// TwinCAT 3 PLC project PLC
// ProgramVersion: 3.1.4023.0
// libraries:
//   Tc2_Standard, * (Beckhoff Automation GmbH)
//   Tc2_System, * (Beckhoff Automation GmbH)
//   Tc2_Utilities, * (Beckhoff Automation GmbH)
//   Tc3_Module, * (Beckhoff Automation GmbH)
// project tree:
//   Encryption/Blowfish/ FB_Blowfish.TcPOU, P_Blowfish.TcPOU
//   / PlcTask.TcTTO
//   POUs/ MAIN.TcPOU
// real-time tasks:
//   TASK PlcTask: cycle T#10ms, priority 20, ADS port 350

CONFIGURATION PLC
    RESOURCE PLC ON TwinCAT3
        TASK PlcTask(INTERVAL := T#10ms, PRIORITY := 20);
        PROGRAM MAIN WITH PlcTask : MAIN;
    END_RESOURCE
END_CONFIGURATION

// ---- POUs/MAIN.TcPOU
PROGRAM MAIN

// Blowfish test
P_Blowfish();

END_PROGRAM

// ---- Encryption/Blowfish/P_Blowfish.TcPOU
(* 
	Encrypting data with the Blowfish algorithm
	More info: https://www.schneier.com/academic/blowfish/

	original code 
	C by Bruce Schneier	https://www.schneier.com/wp-content/uploads/2015/12/bfsh-sch.zip

	TwinCAT code released under MIT license (https://opensource.org/licenses/MIT)
	Kim Robbens (2022) 	
	
	USAGE:
		* The subkeyfile BLOWFISH.DAT should be placed in the TwinCAT default boot folder. 
		  In most cases this is C:\TwinCAT\3.1\Boot.
		* define instance of FB_BlowFish
		* define a secret key, can be any data type, the max length is 56 bytes / 448 bits
		  as defined in the Blowfish specification
		* initialize the FB_Blowfish instance with the necessary parameters  
			- secret key
			- length of the secret key
			- endianness of the system, TRUE: Eg: Intel, FALSE: Eg: Motorola 
*)
PROGRAM P_Blowfish
VAR
	// Blowfish algorithm
	fbBlowFish			: FB_BlowFish;
	
	// Test secret key
	key 				: T_MAXSTRING := 'TESTKEY';
	
	
	
	(********************  UNIT TESTS  ***********************)
	// Test string to encrypt, its length should be a multiple of 4 bytes
	// real size of a string is [15] + NULL character == 16 !!
	sString				: STRING[15] := 'ABCDEFGHIJKLMNO';	
	nStringLengthOK		: DINT;
	// If the length is nok, an error will be returned with the # of exceeding bytes 
	sStringNOK			: STRING[17] := 'ABCD_EFGH_IJKL_MN';
	nStringLengthNOK	: DINT;

	// Test array to encrypt
	byBytes				: ARRAY[0..7] OF BYTE := [16#11,16#12,16#13,16#14,16#15,16#16,16#0,16#0];
	nArrayLengthOK		: DINT;
	
	// Test lreal
	lr					: LREAL := 123.2231; // be aware of binary notation rounding!
	nlr					: DINT;

	// test lint
	li					: LINT := -12123123412345;
	nli					: DINT;	
	(********************  UNIT TESTS  ***********************)
END_VAR

// Make sure the subkey file blowfish.dat is located in the TwinCAT 3 root boot folder
// eg. C:\TwinCAT\3.1\Boot

// Blowfish implementation test
IF fbBlowFish.bInitialized		THEN
	(********************  UNIT TESTS  ***********************)
	// Any datatype can be used to encrypt, 
	// as long as it real length MOD 8 == 0
	// examples below 
	nStringLengthOK 	:= fbBlowFish.encrypt(sString);		// string length is ok
	nStringLengthOK 	:= fbBlowFish.decrypt(sString);
	nStringLengthNOK 	:= fbBlowFish.encrypt(sStringNOK);	// returns the # of extra characters
	nStringLengthNOK 	:= fbBlowFish.decrypt(sStringNOK);
	nArrayLengthOK 		:= fbBlowFish.encrypt(byBytes);		// test bytes array
	nArrayLengthOK 		:= fbBlowFish.decrypt(byBytes);
	nlr 				:= fbBlowFish.encrypt(lr);			// test lreal
	nlr 				:= fbBlowFish.decrypt(lr);
	nli 				:= fbBlowFish.encrypt(li);			// test lint
	nli 				:= fbBlowFish.decrypt(li);	
	(********************  UNIT TESTS  ***********************)
ELSE	// Initializing
	fbBlowFish(SecretKey:=ADR(key), SecretKeyBytes:=len(key), bLittleEndian:=TRUE);	
END_IF

END_PROGRAM

// ---- Encryption/Blowfish/FB_Blowfish.TcPOU
(* 
	Encrypting data with the Blowfish algorithm, more info below

	original code 
	C by Bruce Schneier	https://www.schneier.com/wp-content/uploads/2015/12/bfsh-sch.zip

	TwinCAT code released under MIT license (https://opensource.org/licenses/MIT)
	Kim Robbens (2022) 
	
	<!HARD LIMITATION
	Due to the limitations of codesys memory allocations,
	it is only possible to encrypt datablocks that have a byte length MOD 8 == 0	
	eg STRING[8] is 9 bytes!!
	See example implementation
	HARD LIMITATION!>
*)
{attribute 'hide_all_locals'}
FUNCTION_BLOCK FB_Blowfish
VAR_INPUT
	SecretKey				: POINTER TO BYTE;	// Make sure that the object is a multiple of 4 bytes!
	SecretKeyBytes			: INT;
	bLittleEndian			: BOOL:=TRUE;	(* TRUE: Eg: Intel, FALSE: Eg: Motorola *)
END_VAR
VAR_OUTPUT
	bBusy                   : BOOL; 	(* TRUE => execution in progress, FALSE => execution idle *)
 	bError                  : BOOL; 	(* TRUE => Error, FALSE => No error *)
	bInitialized			: BOOL;		(* TRUE => initialization of the cipher OK *)
 	nErrorId                : UDINT;	(* Error code *)
END_VAR
VAR
	// Internal selftest results
	bSelfTestEncryptionOK	: BOOL;		(* TRUE => internal encryption selftest OK *)
	bSelfTestDecryptionOK	: BOOL;		(* TRUE => internal decryption selftest OK *)	

	// Local Blowfish state enum
	eBF_State				: (	E_BF_Idle, 
								E_BF_FileOpen, E_BF_FileOpening, E_BF_FileIsOpened, 
								E_BF_P_Array_Read, E_BF_P_Array_IsRead, 
								E_BF_S_Boxes_Read, E_BF_S_Boxes_IsRead, 
								E_BF_FileClose, E_BF_FileClosing, E_BF_FileIsClosed,
								E_BF_SelfTest_Encryption, E_BF_SelfTest_Decryption,
								E_BF_Ready, E_BF_Error);		
	// Local error identification
	eErrorID				: ( E_ERR_NoError,
								E_ERR_SelfTest_Encryption,
								E_ERR_DataLength_NOK);
	// File handling
	hSubKeyFile				: UINT := 0;(* File handle of the subkey file *)
	fbFileOpen              : FB_FileOpen;
	fbFileClose             : FB_FileClose;
	fbFileRead              : FB_FileRead;
	// P-Array and S-Boxes
	_P						: ARRAY[0..N+1] OF UDINT; 		// unsigned long P[N + 2];
	_S						: ARRAY[0..3,0..255] OF UDINT; 	// unsigned long S[4][256];
END_VAR
VAR CONSTANT
	MAXKEYBYTES 			: BYTE := 56;          // 448 bits 
	N               		: BYTE := 16;
	subKeyFilename   		: T_MAXSTRING := 'Blowfish.dat';	
END_VAR
(* 
	Encrypting data with the Blowfish algorithm, info below

	Blowfish is unpatented and license-free, and is available free for all uses.

	Source: https://www.embedded.com/encrypting-data-with-the-blowfish-algorithm/

	Generally speaking, encryption algorithms come in two flavors, symmetric and public key. 
	Symmetric algorithms, such as Blowfish, use the same key for encryption and decryption. 
	Like a password, you have to keep the key secret from everyone except the sender and receiver 
	of the message. 

	Blowfish is a symmetric encryption algorithm, meaning that it uses the same secret key 
	to both encrypt and decrypt messages. 
	Blowfish is also a block cipher, meaning that it divides a message up into fixed length blocks 
	during encryption and decryption. The block length for Blowfish is 64 bits; 
	messages that aren't a multiple of eight bytes in size must be padded.

	Blowfish is public domain, and was designed by Bruce Schneier expressly for use in 
	performance-constrained environments such as embedded systems. 
	It has been extensively analyzed and deemed "reasonably secure" by the cryptographic community. 
	Implementation examples are available from several sources, including the one by Bruce Schneier 
	and the one from Paul Kocher that have been used for creating the TwinCAT compatible version. 
	The original code is available for download at https://www.schneier.com/academic/blowfish/download/

	More info: https://www.schneier.com/academic/blowfish/
	
	port of original code 
	C by Bruce Schneier	https://www.schneier.com/wp-content/uploads/2015/12/bfsh-sch.zip
*)

IF NOT bInitialized		THEN
	initialize(SecretKey, SecretKeyBytes, TRUE);
END_IF

METHOD private _busy
bInitialized	:= FALSE;
bError			:= FALSE;
nErrorID		:= TO_UDINT(E_ERR_NoError);
bBusy 			:= TRUE;
END_METHOD

METHOD PRIVATE _done
bError			:= FALSE;
bBusy 			:= FALSE;
nErrorID		:= TO_UDINT(E_ERR_NoError);
bInitialized	:= TRUE;
END_METHOD

METHOD PRIVATE _error
VAR_INPUT
END_VAR
bBusy 			:= FALSE;
bError			:= TRUE;
END_METHOD

METHOD PRIVATE decipher
VAR_INPUT
	xL					: REFERENCE TO UDINT;
	xR					: REFERENCE TO UDINT;
END_VAR
VAR
	temp				: UDINT;
	i					: INT;
END_VAR
FOR i := N+1 TO 2 BY -1 DO		// for (i = N + 1; i > 1; --i)
	xL		:= xL XOR _P[i];
	xR 	:= F(xL) XOR xR;
	// Exchange xL and xR 
	temp 	:= xL;
	xL 	:= xR;
	xR 	:= temp;
END_FOR

// Exchange xL and xR
temp 		:= xL;
xL 		:= xR;
xR 		:= temp;

xR 		:= xR XOR _P[1];
xL 		:= xL XOR _P[0];
END_METHOD

METHOD PUBLIC decrypt 		: DINT
VAR_INPUT
	data					: ANY;	// !!! Only 8 byte multiple sized BYTE arrays !!!
END_VAR
VAR
	dataL					: UDINT;
	dataR					: UDINT;	
	i						: DINT;	
	nMultiples				: DINT;		// Number of blocks of 4 byte
	bEvenMultiples			: BOOL;		// Number of blocks of 4 byte is even
END_VAR
IF bInitialized 			THEN		// Cipher was initialized
	// Blowfish is a 4/8 byte block cipher
	// so first check the length of the data
	// if the data is no multiple of 4, exit with error
	decrypt					:= data.diSize MOD 4;
	IF decrypt = 0 	AND_THEN data.diSize > 0	THEN
		nMultiples			:= data.diSize / 4;				// Number of blocks
		bEvenMultiples		:= nMultiples MOD 2 = 0;		// Even number of blocks
		FOR i := 0 TO nMultiples-1 BY 2 DO
			dataL				:=
			dataR				:= 16#0;
			memcpy(ADR(dataL), ADR(data.pValue[i*4]), 4);
			IF 	i <	nMultiples-1 OR_ELSE bEvenMultiples THEN
				memcpy(ADR(dataR), ADR(data.pValue[(i+1)*4]), 4);
				decipher(dataL, dataR);
				memcpy(ADR(data.pValue[i*4]), ADR(dataL), 4);				
				memcpy(ADR(data.pValue[(i+1)*4]), ADR(dataR), 4);
			ELSE
				decipher(dataL, dataR);
				memcpy(ADR(data.pValue[i*4]), ADR(dataL), 4);				
			END_IF	
		END_FOR
	ELSE
		nErrorId			:= TO_UDINT(E_ERR_DataLength_NOK);
		_error();		
	END_IF  
ELSE
	initialize(SecretKey, SecretKeyBytes, bLittleEndian);
END_IF
END_METHOD

METHOD PRIVATE encipher
VAR_INPUT
	xL					: REFERENCE TO UDINT;
	xR					: REFERENCE TO UDINT;
END_VAR
VAR
	i					: INT;
	temp				: UDINT;
END_VAR
FOR i := 0 TO N-1 DO				// for (i = 0; i < N; ++i)
	xL		:= xL XOR _P[i];
	xR 		:= F(xL) XOR xR;
	// Exchange xL and xR
	temp 	:= xL;
	xL 		:= xR;
	xR 		:= temp;
END_FOR

// Exchange xL and xR 
temp 		:= xL;
xL 			:= xR;
xR 			:= temp;

xR 			:= xR XOR _P[N];		// Xr = Xr ^ _P[N];
xL 			:= xL XOR _P[N + 1];	// Xl = Xl ^ _P[N + 1];
END_METHOD

METHOD PUBLIC encrypt 		: DINT
VAR_INPUT
	data					: ANY;	// !!! Only 8 byte multiple sized BYTE data !!!
END_VAR
VAR
	dataL					: UDINT;
	dataR					: UDINT;	
	i						: DINT;	
	nMultiples				: DINT;		// Number of blocks of 4 byte
	bEvenMultiples			: BOOL;		// Number of blocks of 4 byte is even
END_VAR
IF bInitialized 			THEN		// Cipher was initialized
	// Blowfish is a 4/8 byte block cipher
	// so first check the length of the data
	// if the data is no multiple of 4, exit with error
	encrypt					:= data.diSize MOD 4;
	IF encrypt = 0 	AND_THEN data.diSize > 0	THEN
		nMultiples			:= data.diSize / 4;				// Number of blocks
		bEvenMultiples		:= nMultiples MOD 2 = 0;		// Even number of blocks
		FOR i := 0 TO nMultiples-1 BY 2 DO
			dataL				:=
			dataR				:= 16#0;
			memcpy(ADR(dataL), ADR(data.pValue[i*4]), 4);
			IF 	i <	nMultiples-1 OR_ELSE bEvenMultiples THEN
				memcpy(ADR(dataR), ADR(data.pValue[(i+1)*4]), 4);
				encipher(dataL, dataR);
				memcpy(ADR(data.pValue[i*4]), ADR(dataL), 4);				
				memcpy(ADR(data.pValue[(i+1)*4]), ADR(dataR), 4);
			ELSE
				encipher(dataL, dataR);
				memcpy(ADR(data.pValue[i*4]), ADR(dataL), 4);				
			END_IF	
		END_FOR
	ELSE
		nErrorId			:= TO_UDINT(E_ERR_DataLength_NOK);
		_error();		
	END_IF  
ELSE
	initialize(SecretKey, SecretKeyBytes, bLittleEndian);
END_IF
END_METHOD

METHOD PRIVATE F 			: UDINT
VAR_INPUT
	x						: UDINT;
END_VAR
VAR
	a						: UDINT;
	b						: UDINT;
	c						: UDINT;
	d						: UDINT;
END_VAR
d := x AND 16#00FF;
x := SHR(x,8);			// x >>= 8 ==== x = x >> 8
c := x AND 16#00FF;
x := SHR(x,8);			
b := x AND 16#00FF;
x := SHR(x,8);			
a := x AND 16#00FF;
//y = ((_S[0][a] + _S[1][b]) ^ _S[2][c]) + _S[3][d];
f := _S[0,a] + _S[1,b];
f := f XOR _S[2,c];
f := f + _S[3,d];
END_METHOD

METHOD PRIVATE initialize
VAR_INPUT	
	key						: POINTER TO BYTE;
	keybytes				: INT;
	bLittleEndian			: BOOL:=TRUE;	(* TRUE: Eg: Intel, FALSE: Eg: Motorola *)
END_VAR
VAR
	// Locals
	i						: INT;
	j						: INT;
	k						: INT;
	data					: UDINT;
	dataL					: UDINT;
	dataR					: UDINT;		
END_VAR
CASE eBF_State				OF

	E_BF_Idle:		(* Idle state *)
		_Busy();
		hSubKeyFile			:= 0;
		eBF_State 			:= E_BF_FileOpen;

	E_BF_FileOpen:		(* Open source file *)
         fbFileOpen(bExecute:=FALSE );
         fbFileOpen( 
			sPathName 		:= subKeyFilename,
			nMode 			:= FOPEN_MODEREAD OR FOPEN_MODEBINARY,
            ePath 			:= PATH_BOOTPATH, 
			bExecute 		:= TRUE
			);
		eBF_State 			:= E_BF_FileOpening;

	E_BF_FileOpening:		(* Open source file *)
		fbFileOpen( bExecute := FALSE );
		IF NOT fbFileOpen.bBusy 	THEN
			IF fbFileOpen.bError 	THEN
				nErrorId 	:= fbFileOpen.nErrId;
				eBF_State	:= E_BF_Error;
			ELSE
				hSubKeyFile := fbFileOpen.hFile;
				eBF_State	:= E_BF_FileIsOpened;
			END_IF
		END_IF

	E_BF_FileIsOpened: 	(* Step without specific interaction *)
		eBF_State			:= E_BF_P_Array_Read;

	E_BF_P_Array_Read:
		fbFileRead(bExecute	:= FALSE);	
		fbFileRead(
			hFile			:= hSubKeyFile, 
			pReadBuff		:= ADR(_P), 
			cbReadLen		:= SIZEOF(_P), 
			bExecute		:= TRUE
			);	
		eBF_State 			:= E_BF_P_Array_IsRead;

	E_BF_P_Array_IsRead:
		fbFileRead(bExecute	:= FALSE);	
		IF NOT fbFileRead.bBusy 	THEN
			IF fbFileRead.bError 	THEN
				nErrorId 	:= fbFileRead.nErrId;
				eBF_State	:= E_BF_Error;
			ELSE
				IF bLittleEndian	THEN
					FOR i := 0 TO N+1 DO
						_P[i] := InverseEndian(_P[i]);
					END_FOR
				END_IF				      
				eBF_State	:= E_BF_S_Boxes_Read;
			END_IF
		END_IF
		
	E_BF_S_Boxes_Read:
		fbFileRead(bExecute	:= FALSE);	
		fbFileRead(
			hFile			:= hSubKeyFile, 
			pReadBuff		:= ADR(_S), 
			cbReadLen		:= SIZEOF(_S), 
			bExecute		:= TRUE
			);	
		eBF_State 			:= E_BF_S_Boxes_IsRead;

	E_BF_S_Boxes_IsRead:
		fbFileRead(bExecute	:= FALSE);	
		IF NOT fbFileRead.bBusy 	THEN
			IF fbFileRead.bError 	THEN
				nErrorId 	:= fbFileRead.nErrId;
				eBF_State	:= E_BF_Error;
			ELSE
				IF bLittleEndian	THEN
					FOR i := 0 TO 3 DO
						FOR j := 0 TO 255 DO
							_S[i,j] := InverseEndian(_S[i,j]);							
						END_FOR						
					END_FOR
				END_IF				      
				eBF_State	:= E_BF_Fileclose;
			END_IF
		END_IF

	E_BF_Fileclose:     	(* Close the subkey file *)
	 	fbFileClose( bExecute := FALSE );
		fbFileClose( 
			hFile			:= hSubKeyFile, 
			bExecute		:= TRUE
			);
		eBF_State			:= E_BF_FileClosing;

	E_BF_FileClosing:     (* Closing the subkey file *)
		fbFileClose( bExecute := FALSE );
		IF NOT fbFileClose.bBusy THEN
			IF fbFileClose.bError THEN
				nErrorId 	:= fbFileClose.nErrId;
				eBF_State	:= E_BF_Error;
			ELSE
				hSubKeyFile := 0;
				eBF_State	:= E_BF_FileIsClosed;
			END_IF
		END_IF

	E_BF_FileIsClosed:     (* The subkey file is closed *)
		// Hash the P array with the key
      	j 					:= 0;
      	FOR i := 0 TO N + 1 DO
	 		data := 16#00000000;
	 		FOR k := 0 TO 3 DO
				// Includes the bugfix proposed here
				// https://www.schneier.com/wp-content/uploads/2015/12/blowfish-bug-2.txt
	    		data := SHL(data, 8) OR (key[j] AND 16#FF);
	    		j := j + 1;
	    		IF (j >= keybytes) THEN
	       			j := 0;
				END_IF
			END_FOR
			_P[i] := _P[i] XOR data;
		END_FOR
		dataL 	:= 16#00000000;
      	dataR 	:= 16#00000000;	

		// Encipher the P-array 
      	FOR i := 0 TO N + 1 BY 2 DO
	    	encipher(dataL, dataR);
         	_P[i] := dataL;
         	_P[i + 1] := dataR;
      	END_FOR
		
		// Encipher the S-Boxes
      	FOR i := 0 TO 3 DO
         	FOR j := 0 TO 255 BY 2 DO
	            encipher(dataL, dataR);
            	_S[i,j] 	:= dataL;
            	_S[i,j + 1]	:= dataR;
			END_FOR
		END_FOR		
		eBF_State		:= E_BF_SelfTest_Encryption;

	E_BF_Error: (* Error => Cleanup / retry opening *)
		_error();
		IF (hSubKeyFile <> 0 ) THEN (* Close the subkey file if open*)
			eBF_State		:= E_BF_FileClose; 
	 	ELSE
			eBF_State		:= E_BF_FileOpen;      (* Error, retry open *)
		END_IF

	E_BF_SelfTest_Encryption:	(* Internal self test of the encryption algorithm *)
		dataL				:= 16#1;
		dataR				:= 16#2;	
		encipher(dataL, dataR);
		IF (dataL = 16#DF333FD2 AND dataR = 16#30A71BB4)	THEN
			bSelfTestEncryptionOK 	:= TRUE;
		END_IF
		eBF_State			:= E_BF_SelfTest_Decryption;
		 	
	E_BF_SelfTest_Decryption:	(* Internal self test of the encryption algorithm *)
		dataL				:= 16#DF333FD2;
		dataR				:= 16#30A71BB4;	
		decipher(dataL, dataR);
		IF (dataL = 16#1 AND dataR = 16#2)	THEN
			bSelfTestDecryptionOK 	:= TRUE;
		END_IF
		eBF_State			:= E_BF_Ready;
		 	
	E_BF_Ready:
		IF bSelfTestEncryptionOK AND bSelfTestDecryptionOK		THEN
			_done();
		ELSE
			nErrorId		:= TO_UDINT(E_ERR_SelfTest_Encryption);
			_error();
		END_IF
	ELSE;
		
END_CASE
END_METHOD

METHOD PRIVATE inverseEndian : DWORD
VAR_INPUT
	data		: DWORD;
END_VAR
(*
 data = ((data & 0xFF000000) >> 24) |
	((data & 0x00FF0000) >>  8) |
	((data & 0x0000FF00) <<  8) |
	((data & 0x000000FF) << 24);
*)
InverseEndian := 
	SHR((data AND 16#FF000000), 24) OR
	SHR((data AND 16#00FF0000), 8) OR
	SHL((data AND 16#0000FF00), 8) OR
	SHL((data AND 16#000000FF), 24);
END_METHOD

END_FUNCTION_BLOCK
